// TIA Portal V18 export
// export: Created 2026-03-12T16:04:32.1614085Z, ExportSetting WithDefaults, DisplayName Totally Integrated Automation Portal, DisplayVersion V18 Update 5, DisplayName TIA Portal Openness, DisplayVersion V18 Update 5, DisplayName TIA Portal Version Control Interface, DisplayVersion V18, DisplayName SINAMICS Startdrive Advanced, DisplayVersion V18, DisplayName SINAMICS Startdrive G130, G150, S120, S150, SINAMICS MV, S210, DisplayVersion V18, DisplayName SINAMICS Startdrive G110M, G120, G120C, G120D, G120P, G115D, DisplayVersion V18, DisplayName STEP 7 Professional, DisplayVersion V18 Update 5, DisplayName STEP 7 Safety, DisplayVersion V18, DisplayName WinCC Professional, DisplayVersion V18 Update 5
ORGANIZATION_BLOCK "Resets"   // OB126, LAD, ProgramCycle
TITLE = "Main Program Sweep (Cycle)"
{ S7_Optimized_Access := 'TRUE' }
VERSION : 0.1
// stored: AutoNumber true, IsIECCheckEnabled false, SetENOAutomatically false
   VAR_INPUT
      Initial_Call : Bool;   // Initial call of this OB
      Remanence : Bool;   // =True, if remanent data are available
   END_VAR
   VAR_TEMP   // added for the SCL form of the ladder/FBD networks
      _w1 : Bool;
   END_VAR
BEGIN

REGION Network 1: Reset Aferição (Inversor/Instrumentação)
   // Se o valor do comando de aferição for diferente de 0, um tempo será disparado para que a aferição seja feita, em seguida, os valores de entrada serão zerados
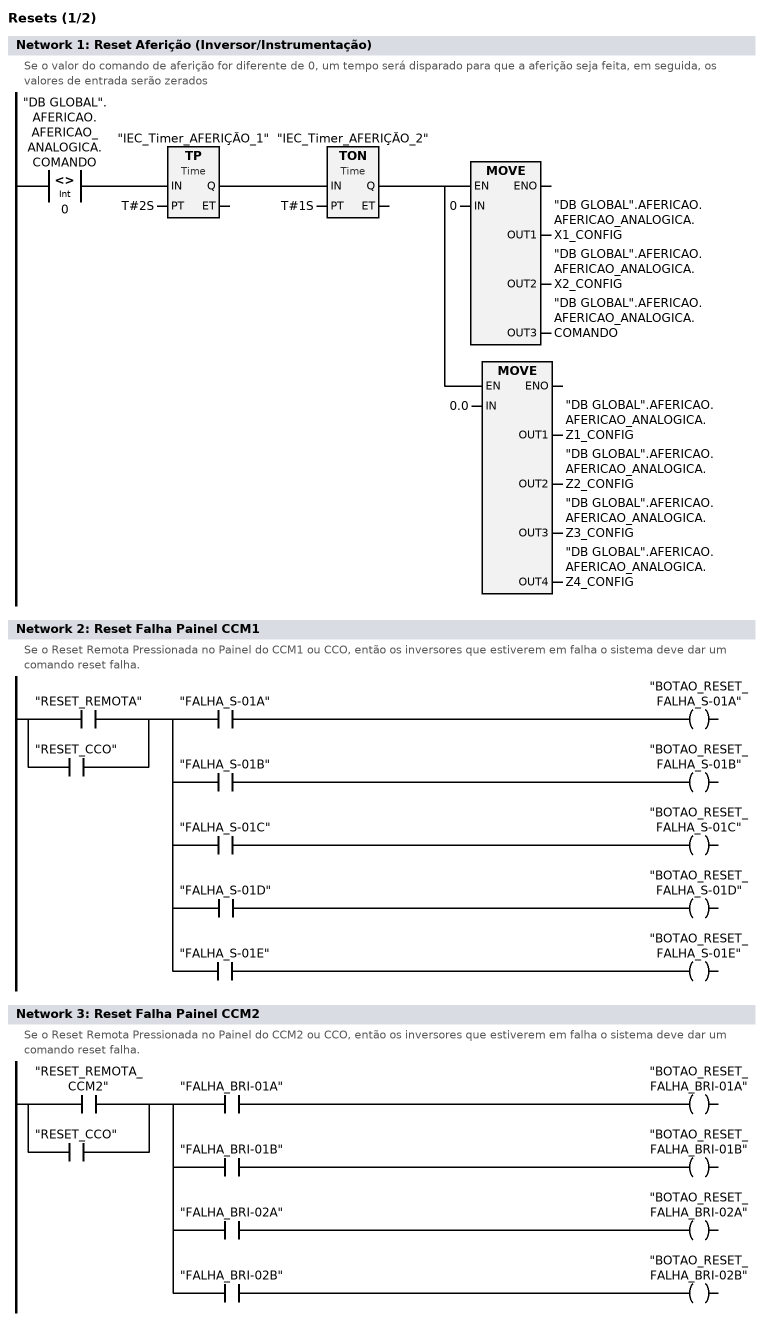
   RUNG wire#powerrail
      { S7_Templates := "SrcType := Int" } NE_Contact(in1 := "DB GLOBAL".AFERICAO.AFERICAO_ANALOGICA.COMANDO, in2 := 0)
      { S7_Templates := "time_type := Time" } "IEC_Timer_AFERIÇÃO_1".TP(pt := T#2S, et =>)
      { S7_Templates := "time_type := Time" } "IEC_Timer_AFERIÇÃO_2".TON(pt := T#1S, et =>)
      wire#w1
      Move(in := 0, out1 => "DB GLOBAL".AFERICAO.AFERICAO_ANALOGICA.X1_CONFIG, out2 => "DB GLOBAL".AFERICAO.AFERICAO_ANALOGICA.X2_CONFIG, out3 => "DB GLOBAL".AFERICAO.AFERICAO_ANALOGICA.COMANDO)
   END_RUNG
   RUNG wire#w1
      Move(in := 0.0, out1 => "DB GLOBAL".AFERICAO.AFERICAO_ANALOGICA.Z1_CONFIG, out2 => "DB GLOBAL".AFERICAO.AFERICAO_ANALOGICA.Z2_CONFIG, out3 => "DB GLOBAL".AFERICAO.AFERICAO_ANALOGICA.Z3_CONFIG, out4 => "DB GLOBAL".AFERICAO.AFERICAO_ANALOGICA.Z4_CONFIG)
   END_RUNG
   // the same network as SCL:
   "IEC_Timer_AFERIÇÃO_1".TP(IN := "DB GLOBAL".AFERICAO.AFERICAO_ANALOGICA.COMANDO <> 0, PT := T#2S);
   "IEC_Timer_AFERIÇÃO_2".TON(IN := "IEC_Timer_AFERIÇÃO_1".Q, PT := T#1S);
   IF "IEC_Timer_AFERIÇÃO_2".Q THEN
       "DB GLOBAL".AFERICAO.AFERICAO_ANALOGICA.X1_CONFIG := 0;
       "DB GLOBAL".AFERICAO.AFERICAO_ANALOGICA.X2_CONFIG := 0;
       "DB GLOBAL".AFERICAO.AFERICAO_ANALOGICA.COMANDO := 0;
       "DB GLOBAL".AFERICAO.AFERICAO_ANALOGICA.Z1_CONFIG := 0.0;
       "DB GLOBAL".AFERICAO.AFERICAO_ANALOGICA.Z2_CONFIG := 0.0;
       "DB GLOBAL".AFERICAO.AFERICAO_ANALOGICA.Z3_CONFIG := 0.0;
       "DB GLOBAL".AFERICAO.AFERICAO_ANALOGICA.Z4_CONFIG := 0.0;
   END_IF;
END_REGION

REGION Network 2: Reset Falha Painel CCM1
   // Se o Reset Remota Pressionada no Painel do CCM1 ou CCO, então os inversores que estiverem em falha o sistema deve dar um comando reset falha.
   RUNG wire#powerrail
      Contact( "RESET_REMOTA" )
      wire#w1
      Contact( "FALHA_S-01A" )
      Coil( "BOTAO_RESET_FALHA_S-01A" )
   END_RUNG
   RUNG wire#powerrail
      Contact( "RESET_CCO" )
   END_RUNG wire#w1
   RUNG wire#w1
      Contact( "FALHA_S-01B" )
      Coil( "BOTAO_RESET_FALHA_S-01B" )
   END_RUNG
   RUNG wire#w1
      Contact( "FALHA_S-01C" )
      Coil( "BOTAO_RESET_FALHA_S-01C" )
   END_RUNG
   RUNG wire#w1
      Contact( "FALHA_S-01D" )
      Coil( "BOTAO_RESET_FALHA_S-01D" )
   END_RUNG
   RUNG wire#w1
      Contact( "FALHA_S-01E" )
      Coil( "BOTAO_RESET_FALHA_S-01E" )
   END_RUNG
   // the same network as SCL:
   #_w1 := "RESET_REMOTA" OR "RESET_CCO";
   "BOTAO_RESET_FALHA_S-01A" := #_w1 AND "FALHA_S-01A";
   "BOTAO_RESET_FALHA_S-01B" := #_w1 AND "FALHA_S-01B";
   "BOTAO_RESET_FALHA_S-01C" := #_w1 AND "FALHA_S-01C";
   "BOTAO_RESET_FALHA_S-01D" := #_w1 AND "FALHA_S-01D";
   "BOTAO_RESET_FALHA_S-01E" := #_w1 AND "FALHA_S-01E";
END_REGION

REGION Network 3: Reset Falha Painel CCM2
   // Se o Reset Remota Pressionada no Painel do CCM2 ou CCO, então os inversores que estiverem em falha o sistema deve dar um comando reset falha.
   RUNG wire#powerrail
      Contact( "RESET_REMOTA_CCM2" )
      wire#w1
      Contact( "FALHA_BRI-01A" )
      Coil( "BOTAO_RESET_FALHA_BRI-01A" )
   END_RUNG
   RUNG wire#powerrail
      Contact( "RESET_CCO" )
   END_RUNG wire#w1
   RUNG wire#w1
      Contact( "FALHA_BRI-01B" )
      Coil( "BOTAO_RESET_FALHA_BRI-01B" )
   END_RUNG
   RUNG wire#w1
      Contact( "FALHA_BRI-02A" )
      Coil( "BOTAO_RESET_FALHA_BRI-02A" )
   END_RUNG
   RUNG wire#w1
      Contact( "FALHA_BRI-02B" )
      Coil( "BOTAO_RESET_FALHA_BRI-02B" )
   END_RUNG
   // the same network as SCL:
   #_w1 := "RESET_REMOTA_CCM2" OR "RESET_CCO";
   "BOTAO_RESET_FALHA_BRI-01A" := #_w1 AND "FALHA_BRI-01A";
   "BOTAO_RESET_FALHA_BRI-01B" := #_w1 AND "FALHA_BRI-01B";
   "BOTAO_RESET_FALHA_BRI-02A" := #_w1 AND "FALHA_BRI-02A";
   "BOTAO_RESET_FALHA_BRI-02B" := #_w1 AND "FALHA_BRI-02B";
END_REGION

REGION Network 4: Reset Reset Painel CCM3
   // Se o Reset Remota Pressionada no Painel do CCM3 ou CCO, então os inversores que estiverem em falha o sistema deve dar um comando reset falha.
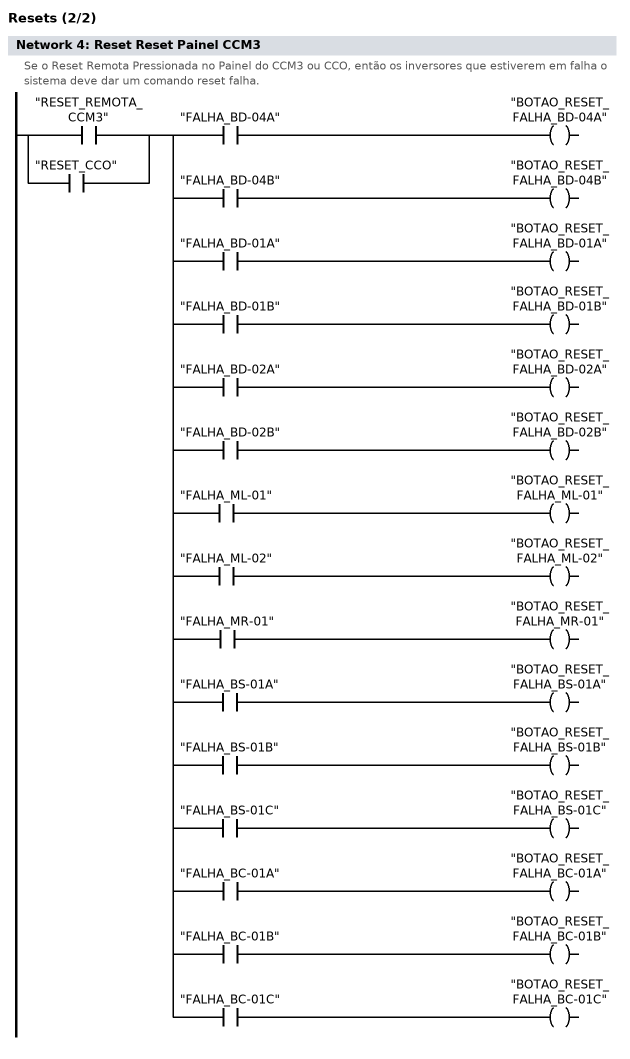
   RUNG wire#powerrail
      Contact( "RESET_REMOTA_CCM3" )
      wire#w1
      Contact( "FALHA_BD-04A" )
      Coil( "BOTAO_RESET_FALHA_BD-04A" )
   END_RUNG
   RUNG wire#powerrail
      Contact( "RESET_CCO" )
   END_RUNG wire#w1
   RUNG wire#w1
      Contact( "FALHA_BD-04B" )
      Coil( "BOTAO_RESET_FALHA_BD-04B" )
   END_RUNG
   RUNG wire#w1
      Contact( "FALHA_BD-01A" )
      Coil( "BOTAO_RESET_FALHA_BD-01A" )
   END_RUNG
   RUNG wire#w1
      Contact( "FALHA_BD-01B" )
      Coil( "BOTAO_RESET_FALHA_BD-01B" )
   END_RUNG
   RUNG wire#w1
      Contact( "FALHA_BD-02A" )
      Coil( "BOTAO_RESET_FALHA_BD-02A" )
   END_RUNG
   RUNG wire#w1
      Contact( "FALHA_BD-02B" )
      Coil( "BOTAO_RESET_FALHA_BD-02B" )
   END_RUNG
   RUNG wire#w1
      Contact( "FALHA_ML-01" )
      Coil( "BOTAO_RESET_FALHA_ML-01" )
   END_RUNG
   RUNG wire#w1
      Contact( "FALHA_ML-02" )
      Coil( "BOTAO_RESET_FALHA_ML-02" )
   END_RUNG
   RUNG wire#w1
      Contact( "FALHA_MR-01" )
      Coil( "BOTAO_RESET_FALHA_MR-01" )
   END_RUNG
   RUNG wire#w1
      Contact( "FALHA_BS-01A" )
      Coil( "BOTAO_RESET_FALHA_BS-01A" )
   END_RUNG
   RUNG wire#w1
      Contact( "FALHA_BS-01B" )
      Coil( "BOTAO_RESET_FALHA_BS-01B" )
   END_RUNG
   RUNG wire#w1
      Contact( "FALHA_BS-01C" )
      Coil( "BOTAO_RESET_FALHA_BS-01C" )
   END_RUNG
   RUNG wire#w1
      Contact( "FALHA_BC-01A" )
      Coil( "BOTAO_RESET_FALHA_BC-01A" )
   END_RUNG
   RUNG wire#w1
      Contact( "FALHA_BC-01B" )
      Coil( "BOTAO_RESET_FALHA_BC-01B" )
   END_RUNG
   RUNG wire#w1
      Contact( "FALHA_BC-01C" )
      Coil( "BOTAO_RESET_FALHA_BC-01C" )
   END_RUNG
   // the same network as SCL:
   #_w1 := "RESET_REMOTA_CCM3" OR "RESET_CCO";
   "BOTAO_RESET_FALHA_BD-04A" := #_w1 AND "FALHA_BD-04A";
   "BOTAO_RESET_FALHA_BD-04B" := #_w1 AND "FALHA_BD-04B";
   "BOTAO_RESET_FALHA_BD-01A" := #_w1 AND "FALHA_BD-01A";
   "BOTAO_RESET_FALHA_BD-01B" := #_w1 AND "FALHA_BD-01B";
   "BOTAO_RESET_FALHA_BD-02A" := #_w1 AND "FALHA_BD-02A";
   "BOTAO_RESET_FALHA_BD-02B" := #_w1 AND "FALHA_BD-02B";
   "BOTAO_RESET_FALHA_ML-01" := #_w1 AND "FALHA_ML-01";
   "BOTAO_RESET_FALHA_ML-02" := #_w1 AND "FALHA_ML-02";
   "BOTAO_RESET_FALHA_MR-01" := #_w1 AND "FALHA_MR-01";
   "BOTAO_RESET_FALHA_BS-01A" := #_w1 AND "FALHA_BS-01A";
   "BOTAO_RESET_FALHA_BS-01B" := #_w1 AND "FALHA_BS-01B";
   "BOTAO_RESET_FALHA_BS-01C" := #_w1 AND "FALHA_BS-01C";
   "BOTAO_RESET_FALHA_BC-01A" := #_w1 AND "FALHA_BC-01A";
   "BOTAO_RESET_FALHA_BC-01B" := #_w1 AND "FALHA_BC-01B";
   "BOTAO_RESET_FALHA_BC-01C" := #_w1 AND "FALHA_BC-01C";
END_REGION
END_ORGANIZATION_BLOCK
